// Mitsubishi GX Works2 project: plc1   PLC: Q03UDV

PROGRAM MAIN
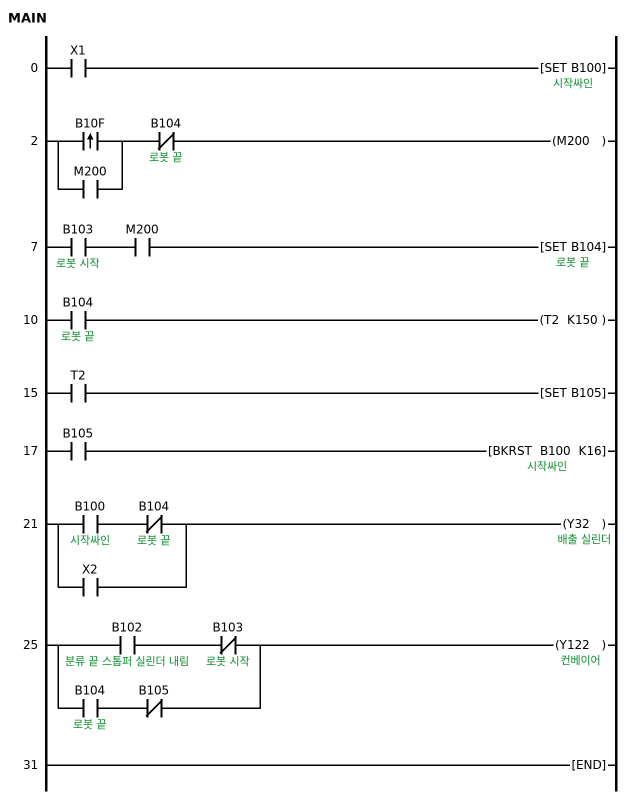
0     LD      X1
      SET     B100  ; 시작싸인
2     LDP     B10F
      OR      M200
      ANI     B104  ; 로봇 끝
      OUT     M200
7     LD      B103  ; 로봇 시작
      AND     M200
      SET     B104  ; 로봇 끝
10    LD      B104  ; 로봇 끝
      OUT     T2 K150
15    LD      T2
      SET     B105
17    LD      B105
      BKRST   B100 K16
21    LD      B100  ; 시작싸인
      ANI     B104  ; 로봇 끝
      OR      X2
      OUT     Y32  ; 배출 실린더
25    LD      B102  ; 분류 끝 스톱퍼 실린더 내림
      ANI     B103  ; 로봇 시작
      LD      B104  ; 로봇 끝
      ANI     B105
      ORB
      OUT     Y122  ; 컨베이어
31    END
END_PROGRAM

// device comments not shown above
B101  ; 스톱퍼 실린더 감지
